FUNCTION_BLOCK StepChain_2
VAR_INPUT
END_VAR
VAR_OUTPUT
END_VAR
VAR
	pSynchPayload : POINTER TO SynchPayload;
	step : UINT;
	timer : TON;
END_VAR

timer(PT:= T#4S);
IF 	pSynchPayload = 0
	THEN
	
	step := 0;
END_IF

CASE step OF
	
	0:
		IF 	fbPayloadCarrier.GetPayload(pSynchPayload,SYNCH_PAYLOAD)
			THEN
			
			step := 10;
		END_IF
		
	10:
	
		IF 	pSynchPayload^.bReleaseRequest
			THEN
			
			pSynchPayload^.bReleaseRequestReceived := TRUE;
			step := 20;
		END_IF
		
	20:
		pSynchPayload^.bReleaseRequestReceived := FALSE;
		timer.IN := TRUE;
		IF  timer.Q
			THEN
			timer.IN := FALSE;
			pSynchPayload^.bRequestAck := TRUE;
			step := 30;
		END_IF
		
	30:	

		IF 	pSynchPayload^.bRequestAckReceived
			THEN
			pSynchPayload^.bRequestAck := FALSE;
			step := 40;
		END_IF
	
	40:;
		
		
END_CASE

END_FUNCTION_BLOCK

(* stored: Version 1.1.0.1, ProductVersion 3.1.4024.2
   POU StepChain_2: Id {81aeb190-d86d-4cd6-b9ec-10df5d75d2cc}, SpecialFunc None *)
